FUNCTION_BLOCK POINT_LIST
  (* Standard: 61499-2 *)
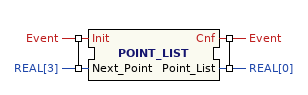
  EVENT_INPUT
    Init WITH Next_Point;
  END_EVENT
  EVENT_OUTPUT
    Cnf WITH Point_List;
  END_EVENT
  VAR_INPUT
    Next_Point : ARRAY [0..2] OF REAL;
  END_VAR
  VAR_OUTPUT
    Point_List : ARRAY [0..-1] OF REAL;
  END_VAR
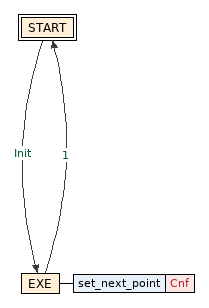
  EC_STATES
    START;
    EXE : set_next_point -> Cnf;
  END_STATES
  EC_TRANSITIONS
    EXE TO START := 1;
    START TO EXE := Init;
  END_TRANSITIONS
  ALGORITHM set_next_point IN Lua:
if type(Point_List) ~= 'table' then
	Point_List = {}
end
if type (Point_List[#Point_List]) == 'table' and Point_List[#Point_List][1] == Next_Point[1] and Point_List[#Point_List][2] == Next_Point[2] and Point_List[#Point_List][3] == Next_Point[3]
	then
else
Point_List[#Point_List +1] = {Next_Point[1], Next_Point[2], Next_Point[3]}
end

--print('\n\nLISTA DE PONTOS\n')
for i, v in ipairs(Point_List) do
	print(v[1], v[2], v[3])
end
  END_ALGORITHM
END_FUNCTION_BLOCK
